INTERFACE IXtsTrack

PROPERTY TrackLength : mc_lreal
GET
END_GET
SET
END_SET
END_PROPERTY

END_INTERFACE

(* stored: Version 1.1.0.1, ProductVersion 3.1.4024.11
   Itf IXtsTrack: Id {b3c6e967-8b31-478f-9f89-976ea42d89c5}
   Property TrackLength: Id {e00364fa-b4dc-4b20-8989-f77a4311510c}
   Get Get: Id {32b4808d-dff1-403b-a19c-9aec12b15f8e}
   Set Set: Id {769c319a-8f8d-4ce1-a3d3-f415e985d23d} *)
